Fanuc KAREL source: kt00513.KL

-- PROVISIONAL review KL for V770-1; original PC SHA256 f4d9a5354c8d82f369a8078a4e02a7fa2817778e0579c52f8f48290bf5631451
-- Incomplete behavior may be omitted. Consult companion uncertainty JSON. Do not deploy.
PROGRAM KT00513
%NOLOCKGROUP
VAR
  OUT : BOOLEAN
-- UNRESOLVED_DECL P1 type=000106
-- UNRESOLVED_DECL P2 type=000101
BEGIN
  -- UNRESOLVED_PC offsets 5-20; opcodes 2E,22,32,35
  -- UNRESOLVED_PC offsets 25-53; opcodes 49,7E,49,AC,23
  -- UNRESOLVED_PC offsets 58-62; opcodes 7F
END KT00513
